PROGRAM MOTOR1
VAR
	iStep : INT ;
	fbRising: R_TRIG;
	fbFalling: F_TRIG;
	bM1DirectionSwitch: BOOL;
	bM1RunOtherDirection: BOOL;
END_VAR

io.M1FaultLight := io.M1FaultStatus;
io.M1RunLight := io.M1RunStatus;

fbRising(CLK:= io.M1StartBtn, Q=> );
fbFalling(CLK:= (io.M1StopBtn), Q=> );

IF fbRising.Q AND io.M1StopBtn THEN 
	//IF bM1DirectionSwitch THEN
		io.M1RunCommand := TRUE;
		//bM1RunOtherDirection := FALSE;
	//ELSE
		//io.M1RunCommand := FALSE;
		//bM1RunOtherDirection := TRUE;
	//END_IF
END_IF

IF fbFalling.Q THEN 
	io.M1RunCommand := FALSE;
END_IF

END_PROGRAM

(* stored: Version 1.1.0.1, ProductVersion 3.1.4022.12
   POU MOTOR1: Id {ef30cc67-8694-4ef0-b9fe-fd04ae26ab04}, SpecialFunc None *)
